{attribute 'qualified_only'}
////{xxxattribute 'strict'}
TYPE E_MODBUS_CMD :
(
	NONE		:=	0,
	INIT		:=	1,
	SEND		:=	2
);
END_TYPE

(* stored: Version 1.1.0.1, ProductVersion 3.1.4022.16
   DUT E_MODBUS_CMD: Id {b001381c-b14d-4ebe-b1a2-8b54c9e0b94b} *)
